// TIA Portal V19 export
VAR_GLOBAL   // PLC tag table "Default tag table"
   Sensor_High_High AT %M0.0 : Bool;
   ACK_Alarm_PB AT %M0.1 : Bool;
   Alarm_Reset_PB AT %M0.2 : Bool;
   AlarmStatus AT %M0.3 : Bool;
   Alarm_Acknowledged AT %M0.4 : Bool;
   Alarm_LED AT %M0.5 : Bool;
   Sensor2_High_High AT %M1.0 : Bool;
   AlarmStatus2 AT %M1.1 : Bool;
   Alarm_Acknowledged2 AT %M0.6 : Bool;
   Alarm_LED2 AT %M0.7 : Bool;
END_VAR
